(* PLC project 未命名, 未知 未命名 1 *)
(* stored: creationDateTime 2021-06-18T18:59:17, modificationDateTime 2021-06-18T20:38:54 *)

PROGRAM hello
  VAR
    button AT %IX0.1 : BOOL;
    lamp AT %QX0.0 : BOOL;
  END_VAR
  VAR
    TOF0 : TOF;
  END_VAR

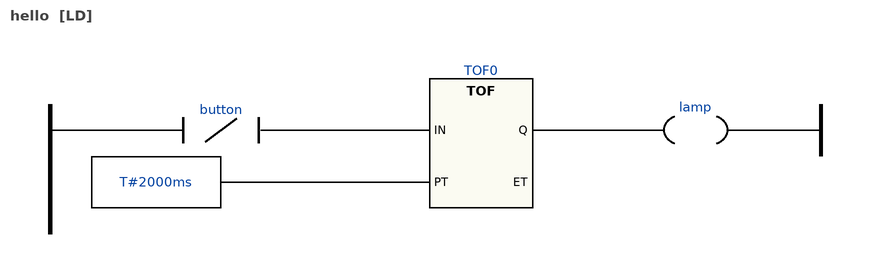
(* LD diagram, written out as Structured Text *)
TOF0(IN := NOT button, PT := T#2000ms);
lamp := TOF0.Q;
END_PROGRAM

CONFIGURATION Config0
  RESOURCE Res0 ON PLC
    TASK task0(INTERVAL := T#20ms, PRIORITY := 0);
    PROGRAM instance0 WITH task0 : hello;
  END_RESOURCE
END_CONFIGURATION
